DATA_BLOCK "F_SystemInfo_DB"
{ S7_Optimized_Access := 'TRUE' }
NAME : F_GLOBDB
VERSION : 0.1
NON_RETAIN
   VAR
      FCCValue : DWord;
   END_VAR


BEGIN

END_DATA_BLOCK

